FUNCTION_BLOCK xPPU_Automatic
VAR CONSTANT
	m_instanceName: STRING := 'xPPU Stamp Workpieces';
END_VAR
VAR_INPUT
	i_ptrErrorManager: POINTER TO ErrorManager;
	i_ptrProcessManager: POINTER TO ProcessManager;
	i_ptrStateTracker: POINTER TO StateTracker;
END_VAR
VAR
	m_stack: xPPU_Stack;
	m_crane: xPPU_Crane;
	m_stamp: xPPU_Stamp;
	m_LSC: xPPU_LSC;
	m_PAC: xPPU_PAC;
	m_PicAlpha: xPPU_PicAlpha;
	m_SSC: xPPU_SSC;
	m_RFC: xPPU_RFC;
	WPConditionOnLSC: BOOL;
END_VAR

VAR
	m_alarm_flags: ARRAY [1..10] OF BOOL := [FALSE, FALSE, FALSE, FALSE, FALSE, FALSE,FALSE, FALSE, FALSE, FALSE]; 
END_VAR

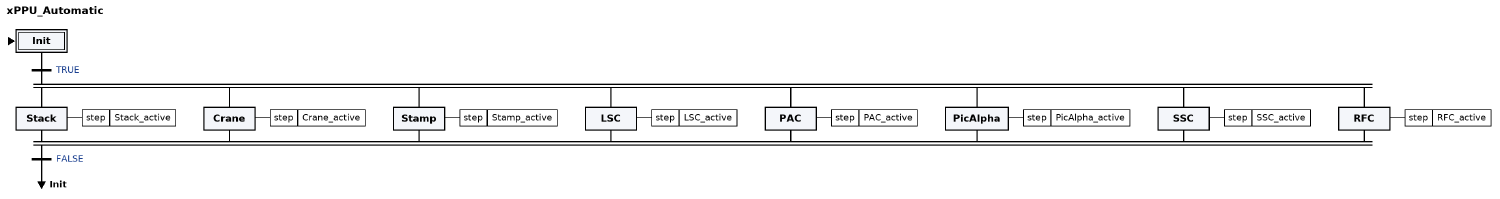
INITIAL_STEP Init:
END_STEP
TRANSITION FROM Init TO (Stack, Crane, Stamp, LSC, PAC, PicAlpha, SSC, RFC)
    := TRUE;
END_TRANSITION
STEP Stack:
    Stack_active(N);  // step action
END_STEP
STEP Crane:
    Crane_active(N);  // step action
END_STEP
STEP Stamp:
    Stamp_active(N);  // step action
END_STEP
STEP LSC:
    LSC_active(N);  // step action
END_STEP
STEP PAC:
    PAC_active(N);  // step action
END_STEP
STEP PicAlpha:
    PicAlpha_active(N);  // step action
END_STEP
STEP SSC:
    SSC_active(N);  // step action
END_STEP
STEP RFC:
    RFC_active(N);  // step action
END_STEP
TRANSITION FROM (Stack, Crane, Stamp, LSC, PAC, PicAlpha, SSC, RFC) TO Init
    := FALSE;
END_TRANSITION

ACTION Crane_active:
m_crane(
	i_error := i_ptrErrorManager, 
	i_process := i_ptrProcessManager,
	i_state := i_ptrStateTracker);
END_ACTION

ACTION LSC_active:
m_LSC(
	i_error := i_ptrErrorManager, 
	i_process := i_ptrProcessManager,
	i_state := i_ptrStateTracker);
END_ACTION

ACTION PAC_active:
m_PAC(
	i_error := i_ptrErrorManager, 
	i_process := i_ptrProcessManager,
	i_state := i_ptrStateTracker);
END_ACTION

ACTION PicAlpha_active:
m_PicAlpha(
	i_error := i_ptrErrorManager, 
	i_process := i_ptrProcessManager,
	i_state := i_ptrStateTracker);
END_ACTION

ACTION RFC_active:
// TODO - this messes up the screwdriver demo! (deactivated for now)

m_RFC(
	i_error := i_ptrErrorManager, 
	i_process := i_ptrProcessManager,
	i_state := i_ptrStateTracker);
END_ACTION

ACTION SSC_active:
m_SSC(
	i_error := i_ptrErrorManager, 
	i_process := i_ptrProcessManager,
	i_state := i_ptrStateTracker);
END_ACTION

ACTION Stack_active:
m_stack(
	i_error := i_ptrErrorManager, 
	i_process := i_ptrProcessManager,
	i_state := i_ptrStateTracker);
END_ACTION

ACTION Stamp_active:
m_stamp(
	i_error := i_ptrErrorManager, 
	i_process := i_ptrProcessManager,
	i_state := i_ptrStateTracker);
END_ACTION

PROPERTY SubSteps : ARRAY [0..2] OF STRING
GET
VAR
	m_tmp: ARRAY [0..2] OF STRING;
END_VAR
m_tmp[0] := TO_STRING(m_stack.SFCCurrentStep);
m_tmp[1] := TO_STRING(m_crane.SFCCurrentStep);
m_tmp[2] := TO_STRING(m_stamp.SFCCurrentStep);
SubSteps := m_tmp;
END_GET
END_PROPERTY

END_FUNCTION_BLOCK

(* stored: Version 1.1.0.1
   POU xPPU_Automatic: Id {d620e1b2-a8f2-4e3a-afca-2ee00cad64e3}, SpecialFunc None
   Action Crane_active: Id {0d2f021e-c58f-45bb-b107-fffe067e5eee}
   Action LSC_active: Id {b236c931-5316-4b36-83eb-f807aaf1c633}
   Action PAC_active: Id {d1b83b7a-3266-4a85-9588-c64bca673b32}
   Action PicAlpha_active: Id {366ca9fc-8dc3-4e6f-901d-c9974e47b618}
   Action RFC_active: Id {0fb9c8ce-6ab9-4507-80a7-7d55b69dded2}
   Action SSC_active: Id {772c08d9-2dd3-47a6-b5d6-133082b04e9a}
   Action Stack_active: Id {78c6b70a-8a87-476e-966b-b2853e06ebc8}
   Action Stamp_active: Id {d03fdec5-852c-4fb4-a233-a46b4cf14a38}
   Property SubSteps: Id {b0f77bfe-7459-40a9-bf5d-eb87cf9040a3}
   Get Get: Id {16f39e7a-4971-432d-8c11-0f9669220f69} *)
